// Mitsubishi GX Works2 project: 工配乙級 第一題   PLC: FX3U/FX3UC

// task Task_01 (event TRUE, interval 0, priority 31): POU_01

PROGRAM POU_01
VAR
  wstep : INT;
  R_TRIG_EMS : R_TRIG;
  unsynced : BOOL;
  TON_SYNC : TON;
END_VAR
M99 := 
Y1 AND Y2 AND Y3 AND Y4 AND Y5 AND 
Y0 AND
Y11 AND Y12 AND Y13 AND

X1 AND X2 AND 
X0 AND 
X11 AND X12 AND
X5 AND X6 AND X7 AND
X15 AND X16 AND X17;

(*PB1 - X1*)						(*PL1 - Y1*)
(*PB2 - X2*)						(*PL2 - Y2*)
(*EMS NC - X0*)				(*PL3 - Y3*)
(*COS 1 - X11*)				(*PL4 - Y4*)
(*COS 2 - X12*)				(*PL5 - Y5*)
(*TH-RY 1 NC - X5*)		(*BZ - Y0*)	
(*TH-RY 2 NC - X6*)		(*MC1 - Y11*)
(*TH-RY 3 NC - X7*)		(*MC2 - Y12*)	
(*MC1 NO - X15*)				(*MC3 - Y13*)	
(*MC2 NO - X16*)
(*MC3 NO - X17*)

IF M8002 THEN
	wstep := 0;
END_IF;

IF wstep <> 60 THEN (*MC 無法同步*)

	(*排空輸送帶*)
	IF X1 AND X0 THEN
		wstep := 1;
	END_IF;
	
	(*EMS*)
	R_TRIG_EMS(_CLK := NOT X0);
	IF R_TRIG_EMS.Q THEN
		wstep := 2;
	END_IF;
	
	(*過載*)
	IF NOT (X5 AND X6 AND X7) THEN
		Y0 := (NOT X12) AND X11;
		SET(TRUE, Y5);
		RST(TRUE, Y11);
		RST(TRUE, Y1);
	END_IF;
	
	IF NOT (X6 AND X7) THEN
		Y0 := (NOT X12) AND X11;
		SET(TRUE, Y5);
		RST(TRUE, Y12);
		RST(TRUE , Y2);
	END_IF;
	
	IF NOT X7 THEN
		Y0 := (NOT X12) AND X11;
		SET(TRUE, Y5);	
		RST(TRUE, Y13);
		RST(TRUE, Y3);
	END_IF;
END_IF;

(*MC無法同步*)
TON_SYNC(IN := (X15 XOR Y11) OR (X16 XOR Y12) OR (X17 XOR Y13), PT := T#2s);
IF TON_SYNC.Q THEN
	wstep := 60;
END_IF;

CASE wstep OF

	0: (*正常模式*)
		ZRST(TRUE, TC250, TC252);
		ZRST(TRUE, Y0, Y17);
		SET(TRUE, Y4);
		Y0 := X12 AND NOT X11;
		IF NOT (X5 AND X6 AND X7) THEN (*過載*)
			wstep := 52;
		END_IF;
		IF X2 THEN (*正常運行*)
			wstep := 20;
		END_IF;
	1: (*排空模式*)
		ZRST(TRUE, TC0, TC2);
		wstep := 30;
	2: (*EMS*)
		ZRST(TRUE, Y0, Y17);
		wstep := 40;	
	3: (*過載*)
		ZRST(TRUE, TC0, TC2);
		IF NOT X7 THEN
			wstep := 52;
		ELSIF NOT X6 THEN
			wstep := 51;
		ELSIF NOT X5 THEN
			wstep := 50;
		END_IF;	
		
	20: (*正常模式*)
		SET(TRUE, Y1);
		SET(TRUE, Y11);
		Y4 := M8013;
		OUT_T(TRUE, TC250, 50);
		IF TS250 OR NOT (X5 AND X6 AND X7) THEN
			wstep := 21;
		END_IF;
	21:
		SET(TRUE, Y2);
		SET(TRUE, Y12);
		Y4 := M8013;
		OUT_T(TRUE, TC251, 100);
		IF TS251 OR NOT (X6 AND X7) THEN
			wstep := 22;
		END_IF;
	22:
		SET(TRUE, Y3);
		SET(TRUE, Y13);
		SET(TRUE, Y4);
		IF NOT (X5 AND X6 AND X7) THEN
			wstep := 3;
		END_IF;
		
	30: (*排空模式*)
		SET(TRUE, Y1);
		SET(TRUE, Y2);
		SET(TRUE, Y3);
		SET(TRUE, Y11);
		SET(TRUE, Y12);
		SET(TRUE, Y13);
		Y4 := M8013;
		Y1 := NOT M8013;
		OUT_T(TRUE, TC0, 50);
		IF TS0 OR NOT (X5 AND X6 AND X7) THEN
			wstep := 31;
		END_IF;
	31:
	 	RST(TRUE, Y1);
		RST(TRUE, Y11);
		Y4 := M8013;
		Y2 := NOT M8013;
		OUT_T(TRUE, TC1, 100);
		IF TS1 OR NOT (X6 AND X7) THEN
			wstep := 32;
		END_IF;
	32:
		RST(TRUE, Y2);
		RST(TRUE, Y12);
		Y4 := M8013;
		Y3 := NOT M8013;
		OUT_T(TRUE, TC2, 50);
		IF TS2 OR NOT X7 THEN
			wstep := 33;
		END_IF;
	33:
		RST(TRUE, Y3);
		RST(TRUE, Y13);
		IF NOT (X5 AND X6 AND X7) THEN
			wstep := 52;
		ELSE
			wstep := 0;		
		END_IF;
			
		
	40: (*EMS*)
		SET(TRUE, Y4);
		Y0 := M8013;
		IF X0 THEN
			wstep := 41;
		END_IF;
	41:
		RST(TRUE, Y0);
		IF X1 THEN
			wstep := 20;
		END_IF;

	50: (*過載*)
		Y2 := M8013; 
		Y4 := NOT M8013;
		OUT_T(TRUE, TC0, 100);
		IF TS0 THEN
			wstep := 51;
		END_IF;
	51:
		RST(TRUE, Y2);
		RST(TRUE, Y12);
		Y3 := M8013; 
		Y4 := NOT M8013;
		OUT_T(TRUE, TC1, 50);
		IF TS1 THEN
			wstep := 52;
		END_IF;
	52:
		RST(TRUE, Y3);
		RST(TRUE, Y13);
		IF X5 AND X6 AND X7 THEN
			wstep := 0;
		END_IF;
	
	(*MC無法同步*)	
	60:
		ZRST(TRUE, Y0, Y17);
END_CASE;
END_PROGRAM
